(* IEC 61131-3 sources: programs/VI-54/VI-54_20171205/VI-54_20171205/Stations/Screen/LseClass170718/Class/GetLimits, 1 file *)

(* ---- GetLimits.st ---- *)
(*!
<Class
	Name               = "GetLimits"
	Revision           = "0.0"
	RealtimeTask       = "false"
	CyclicTask         = "false"
	BackgroundTask     = "true"
	Sigmatek           = "false"
	OSInterface        = "false"
	HighPriority       = "false"
	Automatic          = "false"
	UpdateMode         = "Prescan"
	SharedCommandTable = "true"
	Objectsize         = "(600,480)">
	<Channels>
		<Server Name="AmaxRobot_mm" Visualized="true" Initialize="false" WriteProtected="true" Retentive="false"/>
		<Server Name="AmaxRobot_units" Visualized="true" Initialize="false" WriteProtected="true" Retentive="false"/>
		<Server Name="MaxSpeedBelt_Mmin" Visualized="true" Initialize="false" WriteProtected="true" Retentive="false"/>
		<Server Name="MaxSpeedBelt_units" Visualized="true" Initialize="false" WriteProtected="true" Retentive="false"/>
		<Server Name="SwMaxRas_gr" Visualized="true" Initialize="false" WriteProtected="true" Retentive="false"/>
		<Server Name="SwMaxRas_units" Visualized="true" Initialize="false" WriteProtected="true" Retentive="false"/>
		<Server Name="SwMaxXas_mm" Visualized="true" Initialize="false" WriteProtected="true" Retentive="false"/>
		<Server Name="SwMaxXas_units" Visualized="true" Initialize="false" WriteProtected="true" Retentive="false"/>
		<Server Name="SwMaxYas_mm" Visualized="true" Initialize="false" WriteProtected="true" Retentive="false"/>
		<Server Name="SwMaxYas_units" Visualized="true" Initialize="false" WriteProtected="true" Retentive="false"/>
		<Server Name="SwMaxZas_mm" Visualized="true" Initialize="false" WriteProtected="true" Retentive="false"/>
		<Server Name="SwMaxZas_units" Visualized="true" Initialize="false" WriteProtected="true" Retentive="false"/>
		<Server Name="SwMinRas_gr" Visualized="true" Initialize="false" WriteProtected="true" Retentive="false"/>
		<Server Name="SwMinRas_units" Visualized="true" Initialize="false" WriteProtected="true" Retentive="false"/>
		<Server Name="SwMinXas_mm" Visualized="true" Initialize="false" WriteProtected="true" Retentive="false"/>
		<Server Name="SwMinXas_units" Visualized="true" Initialize="false" WriteProtected="true" Retentive="false"/>
		<Server Name="SwMinYas_mm" Visualized="true" Initialize="false" WriteProtected="true" Retentive="false"/>
		<Server Name="SwMinYas_units" Visualized="true" Initialize="false" WriteProtected="true" Retentive="false"/>
		<Server Name="SwMinZas_mm" Visualized="true" Initialize="false" WriteProtected="true" Retentive="false"/>
		<Server Name="SwMinZas_units" Visualized="true" Initialize="false" WriteProtected="true" Retentive="false"/>
		<Server Name="VmaxRobot_mm" Visualized="true" Initialize="false" WriteProtected="true" Retentive="false"/>
		<Server Name="VmaxRobot_units" Visualized="true" Initialize="false" WriteProtected="true" Retentive="false"/>
		<Client Name="Belt" Required="true" Internal="false"/>
		<Client Name="Ras" Required="true" Internal="false"/>
		<Client Name="Xas" Required="true" Internal="false"/>
		<Client Name="Yas" Required="true" Internal="false"/>
		<Client Name="Zas" Required="true" Internal="false"/>
	</Channels>
</Class>
*)
GetLimits : CLASS
  //Servers:
	SwMaxXas_mm 	: SvrChCmd_DINT;
	SwMaxXas_units 	: SvrCh_DINT;
	SwMinXas_mm 	: SvrCh_DINT;
	SwMinXas_units 	: SvrCh_DINT;
	SwMaxYas_mm 	: SvrCh_DINT;
	SwMaxYas_units 	: SvrCh_DINT;
	SwMinYas_mm 	: SvrCh_DINT;
	SwMinYas_units 	: SvrCh_DINT;
	SwMaxZas_mm 	: SvrCh_DINT;
	SwMaxZas_units 	: SvrCh_DINT;
	SwMinZas_mm 	: SvrCh_DINT;
	SwMinZas_units 	: SvrCh_DINT;
	SwMaxRas_gr 	: SvrCh_DINT;
	SwMaxRas_units 	: SvrCh_DINT;
	SwMinRas_gr 	: SvrCh_DINT;
	SwMinRas_units 	: SvrCh_DINT;
	MaxSpeedBelt_Mmin 	: SvrCh_DINT;
	MaxSpeedBelt_units 	: SvrCh_DINT;
	VmaxRobot_mm 	: SvrCh_DINT;
	VmaxRobot_units 	: SvrCh_DINT;
	AmaxRobot_mm 	: SvrCh_DINT;
	AmaxRobot_units 	: SvrCh_DINT;
  //Clients:
	Xas 	: CltChCmd__LMCAxis;
	Yas 	: CltChCmd__LMCAxis;
	Zas 	: CltChCmd__LMCAxis;
	Ras 	: CltChCmd__LMCAxis;
	Belt 	: CltChCmd__LMCAxis;
  //Variables:
  //Functions:

	FUNCTION VIRTUAL GLOBAL Background
		VAR_INPUT
			EAX 	: UDINT;
		END_VAR
		VAR_OUTPUT
			state (EAX) 	: UDINT;
		END_VAR;
  //Tables:
	FUNCTION @STD
		VAR_OUTPUT
			ret_code	: CONFSTATES;
		END_VAR;
	FUNCTION GLOBAL TAB @CT_;
END_CLASS;

#pragma usingLtd _LMCAxis

FUNCTION VIRTUAL GLOBAL GetLimits::Background
	VAR_INPUT
		EAX 	: UDINT;
	END_VAR
	VAR_OUTPUT
		state (EAX) 	: UDINT;
	END_VAR

  // Xas
  SwMaxXas_units      := Xas.ReadSWEndPos(Mode:=LMCAXIS_RD_SWMAX_APPUNIT); // in units
  SwMinXas_units      := Xas.ReadSWEndPos(Mode:=LMCAXIS_RD_SWMIN_APPUNIT); // in units
  SwMaxXas_mm         := SwMaxXas_units/cIntUnitsTo_mm; // in mm
  SwMinXas_mm         := SwMinXas_units/cIntUnitsTo_mm; // in mm

  // Yas
  SwMaxYas_units      := Yas.ReadSWEndPos(Mode:=LMCAXIS_RD_SWMAX_APPUNIT); // in units
  SwMinYas_units      := Yas.ReadSWEndPos(Mode:=LMCAXIS_RD_SWMIN_APPUNIT); // in units
  SwMaxYas_mm         := SwMaxYas_units/cIntUnitsTo_mm; // in mm
  SwMinYas_mm         := SwMinYas_units/cIntUnitsTo_mm; // in mm

  // Zas
  SwMaxZas_units      := Zas.ReadSWEndPos(Mode:=LMCAXIS_RD_SWMAX_APPUNIT); // in units
  SwMinZas_units      := Zas.ReadSWEndPos(Mode:=LMCAXIS_RD_SWMIN_APPUNIT); // in units
  SwMaxZas_mm         := SwMaxZas_units/cIntUnitsTo_mm; // in mm
  SwMinZas_mm         := SwMinZas_units/cIntUnitsTo_mm; // in mm

  // Ras
  SwMaxRas_units      := Ras.ReadSWEndPos(Mode:=LMCAXIS_RD_SWMAX_APPUNIT); // in units
  SwMinRas_units      := Ras.ReadSWEndPos(Mode:=LMCAXIS_RD_SWMIN_APPUNIT); // in units
  SwMaxRas_gr         := SwMaxRas_units/cIntUnitsTo_mm; // in mm
  SwMinRas_gr         := SwMinRas_units/cIntUnitsTo_mm; // in mm

  // Belt
  MaxSpeedBelt_units  := Belt.ReadParameter(ParNr:=LMCAXIS_PAR_RD_V_MAX, mode:=0); // in units
  MaxSpeedBelt_Mmin   := MaxSpeedBelt_units * 6 / 10000; // M/Min

  // Robot
  if Xas.ReadParameter(ParNr:=LMCAXIS_PAR_RD_V_MAX, mode:=0) <= Yas.ReadParameter(ParNr:=LMCAXIS_PAR_RD_V_MAX, mode:=0) <= Zas.ReadParameter(ParNr:=LMCAXIS_PAR_RD_V_MAX, mode:=0)  then
    VmaxRobot_units := Xas.ReadParameter(ParNr:=LMCAXIS_PAR_RD_V_MAX, mode:=0);
  elsif Yas.ReadParameter(ParNr:=LMCAXIS_PAR_RD_V_MAX, mode:=0) <= Xas.ReadParameter(ParNr:=LMCAXIS_PAR_RD_V_MAX, mode:=0) <= Zas.ReadParameter(ParNr:=LMCAXIS_PAR_RD_V_MAX, mode:=0) then
    VmaxRobot_units := Yas.ReadParameter(ParNr:=LMCAXIS_PAR_RD_V_MAX, mode:=0);
  elsif Zas.ReadParameter(ParNr:=LMCAXIS_PAR_RD_V_MAX, mode:=0) <= Xas.ReadParameter(ParNr:=LMCAXIS_PAR_RD_V_MAX, mode:=0)  <= Yas.ReadParameter(ParNr:=LMCAXIS_PAR_RD_V_MAX, mode:=0) then
    VmaxRobot_units := Zas.ReadParameter(ParNr:=LMCAXIS_PAR_RD_V_MAX, mode:=0);
  else
    VmaxRobot_units := Xas.ReadParameter(ParNr:=LMCAXIS_PAR_RD_V_MAX, mode:=0);
  end_if;
  VmaxRobot_mm := VmaxRobot_units/cIntUnitsTo_mm;

  if Xas.ReadParameter(ParNr:=LMCAXIS_PAR_RD_A_MAX, mode:=0) <= Yas.ReadParameter(ParNr:=LMCAXIS_PAR_RD_A_MAX, mode:=0) <= Zas.ReadParameter(ParNr:=LMCAXIS_PAR_RD_A_MAX, mode:=0)  then
    AmaxRobot_units := Xas.ReadParameter(ParNr:=LMCAXIS_PAR_RD_A_MAX, mode:=0);
  elsif Yas.ReadParameter(ParNr:=LMCAXIS_PAR_RD_A_MAX, mode:=0) <= Xas.ReadParameter(ParNr:=LMCAXIS_PAR_RD_A_MAX, mode:=0) <= Zas.ReadParameter(ParNr:=LMCAXIS_PAR_RD_A_MAX, mode:=0) then
    AmaxRobot_units := Yas.ReadParameter(ParNr:=LMCAXIS_PAR_RD_A_MAX, mode:=0);
  elsif Zas.ReadParameter(ParNr:=LMCAXIS_PAR_RD_A_MAX, mode:=0) <= Xas.ReadParameter(ParNr:=LMCAXIS_PAR_RD_A_MAX, mode:=0)  <= Yas.ReadParameter(ParNr:=LMCAXIS_PAR_RD_A_MAX, mode:=0) then
    AmaxRobot_units := Zas.ReadParameter(ParNr:=LMCAXIS_PAR_RD_A_MAX, mode:=0);
  else
    AmaxRobot_units := Xas.ReadParameter(ParNr:=LMCAXIS_PAR_RD_A_MAX, mode:=0);
  end_if;
  AmaxRobot_mm := AmaxRobot_units/cIntUnitsTo_mm;

	state := READY;

END_FUNCTION
